LIN {X 0,Y 245.189,Z 1176.16,A -85,B 0,C 180,E1 20303.764,E2 20303.764} C_VEL
LIN {X 0,Y 259.827,Z 1145.905,A -85,B 0,C 180,E1 20307.743,E2 20307.743} C_VEL
LIN {X 0,Y 266.312,Z 1129.34,A -85,B 0,C 180,E1 20309.341,E2 20309.341} C_VEL
LIN {X 0,Y 263.727,Z 1110.426,A -85,B 0,C 180,E1 20314.736,E2 20314.736} C_VEL
LIN {X 0,Y 259.355,Z 1093.422,A -85,B 0,C 180,E1 20321.102,E2 20321.102} C_VEL
LIN {X 0,Y 255.054,Z 1081.089,A -85,B 0,C 180,E1 20327.942,E2 20327.942} C_VEL
LIN {X 0,Y 252.604,Z 1073.864,A -85,B 0,C 180,E1 20334.86,E2 20334.86} C_VEL
LIN {X 0,Y 252.397,Z 1073.391,A -85,B 0,C 180,E1 20342.571,E2 20342.571} C_VEL
LIN {X 0,Y 253.413,Z 1075.546,A -85,B 0,C 180,E1 20346.196,E2 20346.196} C_VEL
LIN {X 0,Y 256.742,Z 1083.33,A -85,B 0,C 180,E1 20352.41,E2 20352.41} C_VEL
LIN {X 0,Y 260.858,Z 1093.545,A -85,B 0,C 180,E1 20357.598,E2 20357.598} C_VEL
LIN {X 0,Y 262.032,Z 1131.057,A -85,B 0,C 180,E1 20365.325,E2 20365.325} C_VEL
LIN {X 0,Y 261.485,Z 1139.676,A -85,B 0,C 180,E1 20366.889,E2 20366.889} C_VEL
LIN {X 0,Y 247.883,Z 1174.599,A -85,B 0,C 180,E1 20370.279,E2 20370.279} C_VEL
LIN {X 0,Y 232.476,Z 1205.485,A -85,B 0,C 180,E1 20374.943,E2 20374.943} C_VEL
LIN {X 0,Y 216.883,Z 1231.951,A -85,B 0,C 180,E1 20380.998,E2 20380.998} C_VEL
LIN {X 0,Y 201.876,Z 1255.228,A -85,B 0,C 180,E1 20389.161,E2 20389.161} C_VEL
LIN {X 0,Y 190.362,Z 1273.058,A -85,B 0,C 180,E1 20398.994,E2 20398.994} C_VEL
LIN {X 0,Y 183.865,Z 1285.563,A -85,B 0,C 180,E1 20410.144,E2 20410.144} C_VEL
LIN {X 0,Y 182.005,Z 1292.009,A -85,B 0,C 180,E1 20420.464,E2 20420.464} C_VEL
LIN {X 0,Y 182.159,Z 1294.054,A -85,B 0,C 180,E1 20430.009,E2 20430.009} C_VEL
LIN {X 0,Y 182.027,Z 1292.019,A -85,B 0,C 180,E1 20439.553,E2 20439.553} C_VEL
LIN {X 0,Y 184.068,Z 1285.438,A -85,B 0,C 180,E1 20450.036,E2 20450.036} C_VEL
LIN {X 0,Y 190.629,Z 1273.108,A -85,B 0,C 180,E1 20460.978,E2 20460.978} C_VEL
LIN {X 0,Y 202.939,Z 1254.088,A -85,B 0,C 180,E1 20471.307,E2 20471.307} C_VEL
LIN {X 0,Y 218.493,Z 1230.096,A -85,B 0,C 180,E1 20479.452,E2 20479.452} C_VEL
LIN {X 0,Y 222.82,Z 1224.302,A -85,B 0,C 180,E1 20481.166,E2 20481.166} C_VEL
LIN {X 0,Y 227.633,Z 1220.781,A -85,B 0,C 180,E1 20482.716,E2 20482.716} C_VEL
LIN {X 0,Y 229.232,Z 1219.381,A -85,B 0,C 180,E1 20483.669,E2 20483.669} C_VEL
LIN {X 0,Y 212.52,Z 1224.351,A -85,B 0,C 180,E1 20490.196,E2 20490.196} C_VEL
LIN {X 0,Y 200.093,Z 1226.199,A -85,B 0,C 180,E1 20497.847,E2 20497.847} C_VEL
LIN {X 0,Y 190.04,Z 1223.798,A -85,B 0,C 180,E1 20508.55,E2 20508.55} C_VEL
LIN {X 0,Y 186.162,Z 1216.357,A -85,B 0,C 180,E1 20518.838,E2 20518.838} C_VEL
LIN {X 0,Y 186.218,Z 1204.944,A -85,B 0,C 180,E1 20528.151,E2 20528.151} C_VEL
LIN {X 0,Y 186.799,Z 1200.69,A -85,B 0,C 180,E1 20531.06,E2 20531.06} C_VEL
LIN {X 0,Y 208.406,Z 1192.088,A -85,B 0,C 180,E1 20545.748,E2 20545.748} C_VEL
LIN {X 0,Y 234.94,Z 1181.218,A -85,B 0,C 180,E1 20553.99,E2 20553.99} C_VEL
LIN {X 0,Y 244.119,Z 1176.975,A -85,B 0,C 180,E1 20555.967,E2 20555.967} C_VEL
LIN {X 0,Y 242.991,Z 1180.408,A -85,B 0,C 180,E1 20556.795,E2 20556.795} C_VEL
LIN {X 0,Y 235.158,Z 1193.598,A -85,B 0,C 180,E1 20559.308,E2 20559.308} C_VEL
LIN {X 0,Y 224.981,Z 1205.626,A -85,B 0,C 180,E1 20561.254,E2 20561.254} C_VEL
LIN {X 0,Y 214.6,Z 1216.631,A -85,B 0,C 180,E1 20563.537,E2 20563.537} C_VEL
LIN {X 0,Y 199.114,Z 1236.248,A -85,B 0,C 180,E1 20571.288,E2 20571.288} C_VEL
LIN {X 0,Y 186.349,Z 1251.331,A -85,B 0,C 180,E1 20580.92,E2 20580.92} C_VEL
LIN {X 0,Y 177.863,Z 1261.693,A -85,B 0,C 180,E1 20592.716,E2 20592.716} C_VEL
LIN {X 0,Y 175.408,Z 1265.154,A -85,B 0,C 180,E1 20600.083,E2 20600.083} C_VEL
LIN {X 0,Y 174.379,Z 1266.843,A -85,B 0,C 180,E1 20609.99,E2 20609.99} C_VEL
LIN {X 0,Y 175.404,Z 1265.113,A -85,B 0,C 180,E1 20619.898,E2 20619.898} C_VEL
LIN {X 0,Y 180.566,Z 1258.236,A -85,B 0,C 180,E1 20632.044,E2 20632.044} C_VEL
LIN {X 0,Y 191.47,Z 1245.156,A -85,B 0,C 180,E1 20643.473,E2 20643.473} C_VEL
LIN {X 0,Y 206.248,Z 1227.247,A -85,B 0,C 180,E1 20652.605,E2 20652.605} C_VEL
LIN {X 0,Y 223.911,Z 1203.483,A -85,B 0,C 180,E1 20660.002,E2 20660.002} C_VEL
LIN {X 0,Y 240.85,Z 1176.298,A -85,B 0,C 180,E1 20665.36,E2 20665.36} C_VEL
LIN {X 0,Y 255.839,Z 1146.194,A -85,B 0,C 180,E1 20669.271,E2 20669.271} C_VEL
LIN {X 0,Y 261.365,Z 1131.746,A -85,B 0,C 180,E1 20670.814,E2 20670.814} C_VEL
LIN {X 0,Y 259.219,Z 1113.75,A -85,B 0,C 180,E1 20676.341,E2 20676.341} C_VEL
LIN {X 0,Y 256.051,Z 1099.749,A -85,B 0,C 180,E1 20681.89,E2 20681.89} C_VEL
LIN {X 0,Y 252.505,Z 1087.186,A -85,B 0,C 180,E1 20689.138,E2 20689.138} C_VEL
LIN {X 0,Y 250.859,Z 1081.579,A -85,B 0,C 180,E1 20694.824,E2 20694.824} C_VEL
LIN {X 0,Y 250.784,Z 1081.139,A -85,B 0,C 180,E1 20702.587,E2 20702.587} C_VEL
LIN {X 0,Y 251.644,Z 1083.314,A -85,B 0,C 180,E1 20706.024,E2 20706.024} C_VEL
LIN {X 0,Y 254.452,Z 1090.646,A -85,B 0,C 180,E1 20711.98,E2 20711.98} C_VEL
LIN {X 0,Y 257.709,Z 1099.874,A -85,B 0,C 180,E1 20716.725,E2 20716.725} C_VEL
LIN {X 0,Y 257.468,Z 1137.249,A -85,B 0,C 180,E1 20724.682,E2 20724.682} C_VEL
LIN {X 0,Y 256.636,Z 1142.909,A -85,B 0,C 180,E1 20725.59,E2 20725.59} C_VEL
LIN {X 0,Y 242.493,Z 1176.928,A -85,B 0,C 180,E1 20728.999,E2 20728.999} C_VEL
LIN {X 0,Y 226.617,Z 1207.082,A -85,B 0,C 180,E1 20733.669,E2 20733.669} C_VEL
LIN {X 0,Y 209.266,Z 1234.843,A -85,B 0,C 180,E1 20740.333,E2 20740.333} C_VEL
LIN {X 0,Y 193.272,Z 1257.969,A -85,B 0,C 180,E1 20749.174,E2 20749.174} C_VEL
LIN {X 0,Y 181.334,Z 1275.631,A -85,B 0,C 180,E1 20760.056,E2 20760.056} C_VEL
LIN {X 0,Y 175.727,Z 1286.237,A -85,B 0,C 180,E1 20770.834,E2 20770.834} C_VEL
LIN {X 0,Y 174.128,Z 1291.399,A -85,B 0,C 180,E1 20780.028,E2 20780.028} C_VEL
LIN {X 0,Y 174.282,Z 1293.453,A -85,B 0,C 180,E1 20790.01,E2 20790.01} C_VEL
LIN {X 0,Y 174.15,Z 1291.41,A -85,B 0,C 180,E1 20799.99,E2 20799.99} C_VEL
LIN {X 0,Y 176.589,Z 1284.518,A -85,B 0,C 180,E1 20811.306,E2 20811.306} C_VEL
LIN {X 0,Y 184.769,Z 1270.858,A -85,B 0,C 180,E1 20823.466,E2 20823.466} C_VEL
LIN {X 0,Y 197.693,Z 1252.227,A -85,B 0,C 180,E1 20833.405,E2 20833.405} C_VEL
LIN {X 0,Y 215.557,Z 1227.057,A -85,B 0,C 180,E1 20841.973,E2 20841.973} C_VEL
LIN {X 0,Y 219.744,Z 1224.237,A -85,B 0,C 180,E1 20843.378,E2 20843.378} C_VEL
LIN {X 0,Y 218.871,Z 1224.206,A -85,B 0,C 180,E1 20844.125,E2 20844.125} C_VEL
LIN {X 0,Y 199.055,Z 1228.104,A -85,B 0,C 180,E1 20852.945,E2 20852.945} C_VEL
LIN {X 0,Y 188.026,Z 1227.701,A -85,B 0,C 180,E1 20861.275,E2 20861.275} C_VEL
LIN {X 0,Y 179.987,Z 1222.257,A -85,B 0,C 180,E1 20872.775,E2 20872.775} C_VEL
LIN {X 0,Y 178.093,Z 1211.877,A -85,B 0,C 180,E1 20883.642,E2 20883.642} C_VEL
LIN {X 0,Y 178.335,Z 1208.019,A -85,B 0,C 180,E1 20887.291,E2 20887.291} C_VEL
LIN {X 0,Y 198.763,Z 1199.468,A -85,B 0,C 180,E1 20904.327,E2 20904.327} C_VEL
LIN {X 0,Y 222.559,Z 1190.638,A -85,B 0,C 180,E1 20912.846,E2 20912.846} C_VEL
LIN {X 0,Y 234.82,Z 1185.521,A -85,B 0,C 180,E1 20915.778,E2 20915.778} C_VEL
LIN {X 0,Y 233.722,Z 1188.698,A -85,B 0,C 180,E1 20916.671,E2 20916.671} C_VEL
LIN {X 0,Y 216.238,Z 1214.459,A -85,B 0,C 180,E1 20922.87,E2 20922.87} C_VEL
LIN {X 0,Y 214.6,Z 1216.631,A -85,B 0,C 180,E1 20923.537,E2 20923.537} C_VEL
LIN {X 0,Y 204.086,Z 1226.81,A -85,B 0,C 180,E1 20926.208,E2 20926.208} C_VEL
LIN {X 0,Y 193.765,Z 1235.88,A -85,B 0,C 180,E1 20929.325,E2 20929.325} C_VEL
LIN {X 0,Y 179.406,Z 1251.939,A -85,B 0,C 180,E1 20939.679,E2 20939.679} C_VEL
LIN {X 0,Y 170.286,Z 1262.299,A -85,B 0,C 180,E1 20951.92,E2 20951.92} C_VEL
LIN {X 0,Y 166.738,Z 1266.954,A -85,B 0,C 180,E1 20964.534,E2 20964.534} C_VEL
LIN {X 0,Y 166.766,Z 1266.906,A -85,B 0,C 180,E1 20975.564,E2 20975.564} C_VEL
LIN {X 0,Y 170.295,Z 1262.227,A -85,B 0,C 180,E1 20988.058,E2 20988.058} C_VEL
LIN {X 0,Y 179.427,Z 1251.816,A -85,B 0,C 180,E1 21000.296,E2 21000.296} C_VEL
LIN {X 0,Y 193.837,Z 1235.62,A -85,B 0,C 180,E1 21010.682,E2 21010.682} C_VEL
LIN {X 0,Y 211.006,Z 1214.796,A -85,B 0,C 180,E1 21018.659,E2 21018.659} C_VEL
LIN {X 0,Y 229.31,Z 1188.648,A -85,B 0,C 180,E1 21024.922,E2 21024.922} C_VEL
LIN {X 0,Y 245.601,Z 1159.936,A -85,B 0,C 180,E1 21029.327,E2 21029.327} C_VEL
LIN {X 0,Y 256.523,Z 1135.753,A -85,B 0,C 180,E1 21031.929,E2 21031.929} C_VEL
LIN {X 0,Y 255.032,Z 1118.805,A -85,B 0,C 180,E1 21037.383,E2 21037.383} C_VEL
LIN {X 0,Y 252.373,Z 1104.64,A -85,B 0,C 180,E1 21043.411,E2 21043.411} C_VEL
LIN {X 0,Y 249.75,Z 1093.879,A -85,B 0,C 180,E1 21050.217,E2 21050.217} C_VEL
LIN {X 0,Y 248.747,Z 1089.066,A -85,B 0,C 180,E1 21055.652,E2 21055.652} C_VEL
LIN {X 0,Y 249.002,Z 1088.918,A -85,B 0,C 180,E1 21063.04,E2 21063.04} C_VEL
LIN {X 0,Y 249.794,Z 1091.622,A -85,B 0,C 180,E1 21066.395,E2 21066.395} C_VEL
LIN {X 0,Y 252.674,Z 1099.304,A -85,B 0,C 180,E1 21072.613,E2 21072.613} C_VEL
LIN {X 0,Y 254.53,Z 1105.732,A -85,B 0,C 180,E1 21075.743,E2 21075.743} C_VEL
LIN {X 0,Y 252.921,Z 1141.925,A -85,B 0,C 180,E1 21083.688,E2 21083.688} C_VEL
LIN {X 0,Y 251.045,Z 1148.161,A -85,B 0,C 180,E1 21084.433,E2 21084.433} C_VEL
LIN {X 0,Y 235.684,Z 1182.305,A -85,B 0,C 180,E1 21088.041,E2 21088.041} C_VEL
LIN {X 0,Y 218.408,Z 1212.526,A -85,B 0,C 180,E1 21093.11,E2 21093.11} C_VEL
LIN {X 0,Y 200.991,Z 1238.491,A -85,B 0,C 180,E1 21099.929,E2 21099.929} C_VEL
LIN {X 0,Y 184.644,Z 1260.616,A -85,B 0,C 180,E1 21109.182,E2 21109.182} C_VEL
LIN {X 0,Y 173.275,Z 1276.452,A -85,B 0,C 180,E1 21119.989,E2 21119.989} C_VEL
LIN {X 0,Y 167.402,Z 1287.158,A -85,B 0,C 180,E1 21132.304,E2 21132.304} C_VEL
LIN {X 0,Y 166.257,Z 1290.788,A -85,B 0,C 180,E1 21139.551,E2 21139.551} C_VEL
LIN {X 0,Y 166.389,Z 1292.85,A -85,B 0,C 180,E1 21150.01,E2 21150.01} C_VEL
LIN {X 0,Y 166.279,Z 1290.8,A -85,B 0,C 180,E1 21160.468,E2 21160.468} C_VEL
LIN {X 0,Y 169.039,Z 1283.899,A -85,B 0,C 180,E1 21172.308,E2 21172.308} C_VEL
LIN {X 0,Y 176.763,Z 1271.861,A -85,B 0,C 180,E1 21183.716,E2 21183.716} C_VEL
LIN {X 0,Y 190.692,Z 1253.112,A -85,B 0,C 180,E1 21194.454,E2 21194.454} C_VEL
LIN {X 0,Y 208.282,Z 1229.52,A -85,B 0,C 180,E1 21202.856,E2 21202.856} C_VEL
LIN {X 0,Y 209.933,Z 1228.085,A -85,B 0,C 180,E1 21204.052,E2 21204.052} C_VEL
LIN {X 0,Y 192.381,Z 1230.422,A -85,B 0,C 180,E1 21211.925,E2 21211.925} C_VEL
LIN {X 0,Y 180.743,Z 1229.449,A -85,B 0,C 180,E1 21220.491,E2 21220.491} C_VEL
LIN {X 0,Y 172.225,Z 1223.336,A -85,B 0,C 180,E1 21232.447,E2 21232.447} C_VEL
LIN {X 0,Y 170.257,Z 1215.578,A -85,B 0,C 180,E1 21241.269,E2 21241.269} C_VEL
LIN {X 0,Y 186.699,Z 1207.359,A -85,B 0,C 180,E1 21261.327,E2 21261.327} C_VEL
LIN {X 0,Y 212.387,Z 1198.52,A -85,B 0,C 180,E1 21272.197,E2 21272.197} C_VEL
LIN {X 0,Y 225.811,Z 1193.374,A -85,B 0,C 180,E1 21275.661,E2 21275.661} C_VEL
LIN {X 0,Y 223.008,Z 1198.447,A -85,B 0,C 180,E1 21276.956,E2 21276.956} C_VEL
LIN {X 0,Y 205.444,Z 1221.95,A -85,B 0,C 180,E1 21283.522,E2 21283.522} C_VEL
LIN {X 0,Y 193.765,Z 1235.88,A -85,B 0,C 180,E1 21289.325,E2 21289.325} C_VEL
LIN {X 0,Y 183.692,Z 1243.998,A -85,B 0,C 180,E1 21292.93,E2 21292.93} C_VEL
LIN {X 0,Y 174.018,Z 1250.991,A -85,B 0,C 180,E1 21297.05,E2 21297.05} C_VEL
LIN {X 0,Y 164.217,Z 1261.318,A -85,B 0,C 180,E1 21308.423,E2 21308.423} C_VEL
LIN {X 0,Y 159.862,Z 1266.359,A -85,B 0,C 180,E1 21319.107,E2 21319.107} C_VEL
LIN {X 0,Y 158.63,Z 1268.045,A -85,B 0,C 180,E1 21329.989,E2 21329.989} C_VEL
LIN {X 0,Y 159.855,Z 1266.319,A -85,B 0,C 180,E1 21340.872,E2 21340.872} C_VEL
LIN {X 0,Y 165.373,Z 1259.988,A -85,B 0,C 180,E1 21353.343,E2 21353.343} C_VEL
LIN {X 0,Y 176.842,Z 1248.03,A -85,B 0,C 180,E1 21365.158,E2 21365.158} C_VEL
LIN {X 0,Y 192.75,Z 1230.808,A -85,B 0,C 180,E1 21374.787,E2 21374.787} C_VEL
LIN {X 0,Y 210.471,Z 1209.398,A -85,B 0,C 180,E1 21382.05,E2 21382.05} C_VEL
LIN {X 0,Y 229.446,Z 1182.101,A -85,B 0,C 180,E1 21387.85,E2 21387.85} C_VEL
LIN {X 0,Y 246.322,Z 1151.212,A -85,B 0,C 180,E1 21392.003,E2 21392.003} C_VEL
LIN {X 0,Y 251.68,Z 1138.595,A -85,B 0,C 180,E1 21393.424,E2 21393.424} C_VEL
LIN {X 0,Y 250.651,Z 1121.653,A -85,B 0,C 180,E1 21399.288,E2 21399.288} C_VEL
LIN {X 0,Y 248.464,Z 1107.88,A -85,B 0,C 180,E1 21405.942,E2 21405.942} C_VEL
LIN {X 0,Y 246.888,Z 1100.12,A -85,B 0,C 180,E1 21411.765,E2 21411.765} C_VEL
LIN {X 0,Y 246.49,Z 1096.612,A -85,B 0,C 180,E1 21415.798,E2 21415.798} C_VEL
LIN {X 0,Y 246.762,Z 1096.421,A -85,B 0,C 180,E1 21422.629,E2 21422.629} C_VEL
LIN {X 0,Y 247.472,Z 1099.22,A -85,B 0,C 180,E1 21426.236,E2 21426.236} C_VEL
LIN {X 0,Y 249.649,Z 1105.719,A -85,B 0,C 180,E1 21431.605,E2 21431.605} C_VEL
LIN {X 0,Y 251.154,Z 1111.895,A -85,B 0,C 180,E1 21434.84,E2 21434.84} C_VEL
LIN {X 0,Y 248.303,Z 1146.097,A -85,B 0,C 180,E1 21442.572,E2 21442.572} C_VEL
LIN {X 0,Y 232.505,Z 1180.722,A -85,B 0,C 180,E1 21446.145,E2 21446.145} C_VEL
LIN {X 0,Y 215.352,Z 1209.958,A -85,B 0,C 180,E1 21450.877,E2 21450.877} C_VEL
LIN {X 0,Y 197.136,Z 1236.072,A -85,B 0,C 180,E1 21457.503,E2 21457.503} C_VEL
LIN {X 0,Y 179.845,Z 1258.353,A -85,B 0,C 180,E1 21466.587,E2 21466.587} C_VEL
LIN {X 0,Y 166.334,Z 1275.657,A -85,B 0,C 180,E1 21478.418,E2 21478.418} C_VEL
LIN {X 0,Y 159.887,Z 1286.096,A -85,B 0,C 180,E1 21490.695,E2 21490.695} C_VEL
LIN {X 0,Y 158.393,Z 1290.177,A -85,B 0,C 180,E1 21499.026,E2 21499.026} C_VEL
LIN {X 0,Y 158.511,Z 1292.249,A -85,B 0,C 180,E1 21510.011,E2 21510.011} C_VEL
LIN {X 0,Y 158.417,Z 1290.189,A -85,B 0,C 180,E1 21520.994,E2 21520.994} C_VEL
LIN {X 0,Y 161.528,Z 1283.279,A -85,B 0,C 180,E1 21533.405,E2 21533.405} C_VEL
LIN {X 0,Y 169.964,Z 1271.234,A -85,B 0,C 180,E1 21545.26,E2 21545.26} C_VEL
LIN {X 0,Y 184.925,Z 1252.491,A -85,B 0,C 180,E1 21556.234,E2 21556.234} C_VEL
LIN {X 0,Y 200.873,Z 1231.575,A -85,B 0,C 180,E1 21563.994,E2 21563.994} C_VEL
LIN {X 0,Y 179.115,Z 1232.266,A -85,B 0,C 180,E1 21575.087,E2 21575.087} C_VEL
LIN {X 0,Y 167.187,Z 1227.702,A -85,B 0,C 180,E1 21586.959,E2 21586.959} C_VEL
LIN {X 0,Y 163.61,Z 1223.156,A -85,B 0,C 180,E1 21594.707,E2 21594.707} C_VEL
LIN {X 0,Y 184.744,Z 1211.533,A -85,B 0,C 180,E1 21624.103,E2 21624.103} C_VEL
LIN {X 0,Y 212.713,Z 1202.262,A -85,B 0,C 180,E1 21634.575,E2 21634.575} C_VEL
LIN {X 0,Y 216.482,Z 1200.929,A -85,B 0,C 180,E1 21635.529,E2 21635.529} C_VEL
LIN {X 0,Y 199.29,Z 1223.447,A -85,B 0,C 180,E1 21642.195,E2 21642.195} C_VEL
LIN {X 0,Y 183.326,Z 1241.297,A -85,B 0,C 180,E1 21650.349,E2 21650.349} C_VEL
LIN {X 0,Y 174.018,Z 1250.991,A -85,B 0,C 180,E1 21657.05,E2 21657.05} C_VEL
LIN {X 0,Y 165.048,Z 1256.934,A -85,B 0,C 180,E1 21661.74,E2 21661.74} C_VEL
LIN {X 0,Y 157.034,Z 1261.713,A -85,B 0,C 180,E1 21667.034,E2 21667.034} C_VEL
LIN {X 0,Y 152.089,Z 1266.964,A -85,B 0,C 180,E1 21678.543,E2 21678.543} C_VEL
LIN {X 0,Y 150.759,Z 1268.646,A -85,B 0,C 180,E1 21689.989,E2 21689.989} C_VEL
LIN {X 0,Y 152.081,Z 1266.924,A -85,B 0,C 180,E1 21701.435,E2 21701.435} C_VEL
LIN {X 0,Y 157.886,Z 1260.8,A -85,B 0,C 180,E1 21714.181,E2 21714.181} C_VEL
LIN {X 0,Y 170.386,Z 1248.638,A -85,B 0,C 180,E1 21726.702,E2 21726.702} C_VEL
LIN {X 0,Y 187.178,Z 1231.415,A -85,B 0,C 180,E1 21736.505,E2 21736.505} C_VEL
LIN {X 0,Y 206.521,Z 1208.947,A -85,B 0,C 180,E1 21744.083,E2 21744.083} C_VEL
LIN {X 0,Y 226.033,Z 1181.588,A -85,B 0,C 180,E1 21749.725,E2 21749.725} C_VEL
LIN {X 0,Y 242.637,Z 1151.967,A -85,B 0,C 180,E1 21753.632,E2 21753.632} C_VEL
LIN {X 0,Y 246.974,Z 1142.389,A -85,B 0,C 180,E1 21754.68,E2 21754.68} C_VEL
LIN {X 0,Y 246.55,Z 1125.822,A -85,B 0,C 180,E1 21760.795,E2 21760.795} C_VEL
LIN {X 0,Y 244.976,Z 1112.678,A -85,B 0,C 180,E1 21767.709,E2 21767.709} C_VEL
LIN {X 0,Y 244.18,Z 1104.268,A -85,B 0,C 180,E1 21775.058,E2 21775.058} C_VEL
LIN {X 0,Y 244.112,Z 1103.348,A -85,B 0,C 180,E1 21780.001,E2 21780.001} C_VEL
LIN {X 0,Y 244.781,Z 1105.243,A -85,B 0,C 180,E1 21784.697,E2 21784.697} C_VEL
LIN {X 0,Y 246.87,Z 1113.425,A -85,B 0,C 180,E1 21791.54,E2 21791.54} C_VEL
LIN {X 0,Y 247.813,Z 1116.958,A -85,B 0,C 180,E1 21793.604,E2 21793.604} C_VEL
LIN {X 0,Y 243.764,Z 1149.572,A -85,B 0,C 180,E1 21801.198,E2 21801.198} C_VEL
LIN {X 0,Y 227.344,Z 1183.103,A -85,B 0,C 180,E1 21804.713,E2 21804.713} C_VEL
LIN {X 0,Y 209.921,Z 1211.287,A -85,B 0,C 180,E1 21809.368,E2 21809.368} C_VEL
LIN {X 0,Y 190.906,Z 1237.147,A -85,B 0,C 180,E1 21816.103,E2 21816.103} C_VEL
LIN {X 0,Y 172.532,Z 1259.362,A -85,B 0,C 180,E1 21825.609,E2 21825.609} C_VEL
LIN {X 0,Y 159.501,Z 1274.907,A -85,B 0,C 180,E1 21836.755,E2 21836.755} C_VEL
LIN {X 0,Y 152.238,Z 1285.475,A -85,B 0,C 180,E1 21849.683,E2 21849.683} C_VEL
LIN {X 0,Y 150.544,Z 1289.566,A -85,B 0,C 180,E1 21858.446,E2 21858.446} C_VEL
LIN {X 0,Y 150.618,Z 1291.647,A -85,B 0,C 180,E1 21870.011,E2 21870.011} C_VEL
LIN {X 0,Y 150.595,Z 1289.581,A -85,B 0,C 180,E1 21881.572,E2 21881.572} C_VEL
LIN {X 0,Y 154.087,Z 1282.658,A -85,B 0,C 180,E1 21894.608,E2 21894.608} C_VEL
LIN {X 0,Y 163.325,Z 1270.61,A -85,B 0,C 180,E1 21906.924,E2 21906.924} C_VEL
LIN {X 0,Y 179.675,Z 1251.451,A -85,B 0,C 180,E1 21918.315,E2 21918.315} C_VEL
LIN {X 0,Y 191.17,Z 1237.393,A -85,B 0,C 180,E1 21923.743,E2 21923.743} C_VEL
LIN {X 0,Y 191.403,Z 1236.168,A -85,B 0,C 180,E1 21924.383,E2 21924.383} C_VEL
LIN {X 0,Y 166.271,Z 1232.825,A -85,B 0,C 180,E1 21938.714,E2 21938.714} C_VEL
LIN {X 0,Y 172.135,Z 1218.899,A -85,B 0,C 180,E1 21980.525,E2 21980.525} C_VEL
LIN {X 0,Y 206.98,Z 1208.549,A -85,B 0,C 180,E1 21995.676,E2 21995.676} C_VEL
LIN {X 0,Y 188.21,Z 1230.468,A -85,B 0,C 180,E1 22002.967,E2 22002.967} C_VEL
LIN {X 0,Y 171.707,Z 1247.39,A -85,B 0,C 180,E1 22012.269,E2 22012.269} C_VEL
LIN {X 0,Y 159.314,Z 1259.468,A -85,B 0,C 180,E1 22023.79,E2 22023.79} C_VEL
LIN {X 0,Y 157.034,Z 1261.713,A -85,B 0,C 180,E1 22027.034,E2 22027.034} C_VEL
LIN {X 0,Y 152.147,Z 1264.589,A -85,B 0,C 180,E1 22031.423,E2 22031.423} C_VEL
LIN {X 0,Y 144.275,Z 1267.687,A -85,B 0,C 180,E1 22038.394,E2 22038.394} C_VEL
LIN {X 0,Y 143.942,Z 1267.845,A -85,B 0,C 180,E1 22039.258,E2 22039.258} C_VEL
LIN {X 0,Y 142.879,Z 1269.247,A -85,B 0,C 180,E1 22049.988,E2 22049.988} C_VEL
LIN {X 0,Y 144.338,Z 1267.528,A -85,B 0,C 180,E1 22062.058,E2 22062.058} C_VEL
LIN {X 0,Y 151.066,Z 1261.049,A -85,B 0,C 180,E1 22075.979,E2 22075.979} C_VEL
LIN {X 0,Y 163.868,Z 1249.429,A -85,B 0,C 180,E1 22088.23,E2 22088.23} C_VEL
LIN {X 0,Y 182.191,Z 1231.606,A -85,B 0,C 180,E1 22098.505,E2 22098.505} C_VEL
LIN {X 0,Y 202.17,Z 1209.308,A -85,B 0,C 180,E1 22105.971,E2 22105.971} C_VEL
LIN {X 0,Y 222.848,Z 1181.069,A -85,B 0,C 180,E1 22111.665,E2 22111.665} C_VEL
LIN {X 0,Y 239.933,Z 1151.141,A -85,B 0,C 180,E1 22115.476,E2 22115.476} C_VEL
LIN {X 0,Y 242.38,Z 1145.603,A -85,B 0,C 180,E1 22116.201,E2 22116.201} C_VEL
LIN {X 0,Y 242.5,Z 1131.082,A -85,B 0,C 180,E1 22121.874,E2 22121.874} C_VEL
LIN {X 0,Y 241.778,Z 1119.443,A -85,B 0,C 180,E1 22128.298,E2 22128.298} C_VEL
LIN {X 0,Y 241.447,Z 1112.003,A -85,B 0,C 180,E1 22135.002,E2 22135.002} C_VEL
LIN {X 0,Y 241.542,Z 1110.826,A -85,B 0,C 180,E1 22140.001,E2 22140.001} C_VEL
LIN {X 0,Y 242.11,Z 1112.508,A -85,B 0,C 180,E1 22144.329,E2 22144.329} C_VEL
LIN {X 0,Y 243.898,Z 1121.412,A -85,B 0,C 180,E1 22151.682,E2 22151.682} C_VEL
LIN {X 0,Y 244.152,Z 1124.422,A -85,B 0,C 180,E1 22153.071,E2 22153.071} C_VEL
LIN {X 0,Y 239.703,Z 1151.507,A -85,B 0,C 180,E1 22159.538,E2 22159.538} C_VEL
LIN {X 0,Y 222.574,Z 1185.04,A -85,B 0,C 180,E1 22163.16,E2 22163.16} C_VEL
LIN {X 0,Y 203.297,Z 1214.544,A -85,B 0,C 180,E1 22168.183,E2 22168.183} C_VEL
LIN {X 0,Y 182.848,Z 1240.489,A -85,B 0,C 180,E1 22175.422,E2 22175.422} C_VEL
LIN {X 0,Y 164.862,Z 1260.757,A -85,B 0,C 180,E1 22184.829,E2 22184.829} C_VEL
LIN {X 0,Y 151.259,Z 1275.954,A -85,B 0,C 180,E1 22196.734,E2 22196.734} C_VEL
LIN {X 0,Y 144.011,Z 1285.962,A -85,B 0,C 180,E1 22210.568,E2 22210.568} C_VEL
LIN {X 0,Y 142.346,Z 1290.459,A -85,B 0,C 180,E1 22223.926,E2 22223.926} C_VEL
LIN {X 0,Y 142.719,Z 1291.044,A -85,B 0,C 180,E1 22230.012,E2 22230.012} C_VEL
LIN {X 0,Y 142.748,Z 1288.97,A -85,B 0,C 180,E1 22242.218,E2 22242.218} C_VEL
LIN {X 0,Y 146.687,Z 1282.035,A -85,B 0,C 180,E1 22255.939,E2 22255.939} C_VEL
LIN {X 0,Y 157.741,Z 1269.013,A -85,B 0,C 180,E1 22269.53,E2 22269.53} C_VEL
LIN {X 0,Y 175.278,Z 1249.74,A -85,B 0,C 180,E1 22280.807,E2 22280.807} C_VEL
LIN {X 0,Y 182.492,Z 1240.72,A -85,B 0,C 180,E1 22284.633,E2 22284.633} C_VEL
LIN {X 0,Y 155.611,Z 1236.116,A -85,B 0,C 180,E1 22303.087,E2 22303.087} C_VEL
LIN {X 0,Y 169.698,Z 1222.695,A -85,B 0,C 180,E1 22343.586,E2 22343.586} C_VEL
LIN {X 0,Y 196.981,Z 1214.875,A -85,B 0,C 180,E1 22355.045,E2 22355.045} C_VEL
LIN {X 0,Y 193.49,Z 1219.675,A -85,B 0,C 180,E1 22356.912,E2 22356.912} C_VEL
LIN {X 0,Y 173.323,Z 1240.642,A -85,B 0,C 180,E1 22365.837,E2 22365.837} C_VEL
LIN {X 0,Y 157.722,Z 1255.028,A -85,B 0,C 180,E1 22376.61,E2 22376.61} C_VEL
LIN {X 0,Y 147.832,Z 1264.113,A -85,B 0,C 180,E1 22389.055,E2 22389.055} C_VEL
LIN {X 0,Y 143.942,Z 1267.845,A -85,B 0,C 180,E1 22399.258,E2 22399.258} C_VEL
LIN {X 0,Y 140.501,Z 1269.085,A -85,B 0,C 180,E1 22404.328,E2 22404.328} C_VEL
LIN {X 0,Y 134.969,Z 1269.615,A -85,B 0,C 180,E1 22413.208,E2 22413.208} C_VEL
LIN {X 0,Y 137.544,Z 1267.205,A -85,B 0,C 180,E1 22425.907,E2 22425.907} C_VEL
LIN {X 0,Y 146.933,Z 1259.116,A -85,B 0,C 180,E1 22440.885,E2 22440.885} C_VEL
LIN {X 0,Y 161.652,Z 1246.54,A -85,B 0,C 180,E1 22452.58,E2 22452.58} C_VEL
LIN {X 0,Y 181.356,Z 1227.92,A -85,B 0,C 180,E1 22462.216,E2 22462.216} C_VEL
LIN {X 0,Y 202.141,Z 1204.714,A -85,B 0,C 180,E1 22469.134,E2 22469.134} C_VEL
LIN {X 0,Y 222.14,Z 1177.196,A -85,B 0,C 180,E1 22474.155,E2 22474.155} C_VEL
LIN {X 0,Y 237.837,Z 1149.178,A -85,B 0,C 180,E1 22477.626,E2 22477.626} C_VEL
LIN {X 0,Y 238.482,Z 1135.322,A -85,B 0,C 180,E1 22483.456,E2 22483.456} C_VEL
LIN {X 0,Y 238.316,Z 1124.631,A -85,B 0,C 180,E1 22489.973,E2 22489.973} C_VEL
LIN {X 0,Y 238.487,Z 1118.808,A -85,B 0,C 180,E1 22496.373,E2 22496.373} C_VEL
LIN {X 0,Y 238.695,Z 1118.181,A -85,B 0,C 180,E1 22500.001,E2 22500.001} C_VEL
LIN {X 0,Y 239.151,Z 1119.336,A -85,B 0,C 180,E1 22503.618,E2 22503.618} C_VEL
LIN {X 0,Y 240.466,Z 1127.7,A -85,B 0,C 180,E1 22510.851,E2 22510.851} C_VEL
LIN {X 0,Y 240.406,Z 1130.835,A -85,B 0,C 180,E1 22512.231,E2 22512.231} C_VEL
LIN {X 0,Y 235.396,Z 1154.888,A -85,B 0,C 180,E1 22518.123,E2 22518.123} C_VEL
LIN {X 0,Y 217.201,Z 1188.248,A -85,B 0,C 180,E1 22521.701,E2 22521.701} C_VEL
LIN {X 0,Y 196.658,Z 1217.658,A -85,B 0,C 180,E1 22526.928,E2 22526.928} C_VEL
LIN {X 0,Y 176.654,Z 1241.573,A -85,B 0,C 180,E1 22533.894,E2 22533.894} C_VEL
LIN {X 0,Y 157.206,Z 1262.15,A -85,B 0,C 180,E1 22543.966,E2 22543.966} C_VEL
LIN {X 0,Y 143.248,Z 1276.714,A -85,B 0,C 180,E1 22556.436,E2 22556.436} C_VEL
LIN {X 0,Y 136.068,Z 1285.904,A -85,B 0,C 180,E1 22570.579,E2 22570.579} C_VEL
LIN {X 0,Y 134.439,Z 1289.851,A -85,B 0,C 180,E1 22583.568,E2 22583.568} C_VEL
LIN {X 0,Y 134.824,Z 1290.441,A -85,B 0,C 180,E1 22590.012,E2 22590.012} C_VEL
LIN {X 0,Y 134.914,Z 1288.358,A -85,B 0,C 180,E1 22602.94,E2 22602.94} C_VEL
LIN {X 0,Y 139.379,Z 1281.422,A -85,B 0,C 180,E1 22617.395,E2 22617.395} C_VEL
LIN {X 0,Y 151.197,Z 1268.698,A -85,B 0,C 180,E1 22631.244,E2 22631.244} C_VEL
LIN {X 0,Y 168.526,Z 1250.931,A -85,B 0,C 180,E1 22642.155,E2 22642.155} C_VEL
LIN {X 0,Y 172.973,Z 1246.131,A -85,B 0,C 180,E1 22644.254,E2 22644.254} C_VEL
LIN {X 0,Y 173.089,Z 1244.848,A -85,B 0,C 180,E1 22645.202,E2 22645.202} C_VEL
LIN {X 0,Y 146.179,Z 1239.056,A -85,B 0,C 180,E1 22668.084,E2 22668.084} C_VEL
LIN {X 0,Y 167.723,Z 1226.36,A -85,B 0,C 180,E1 22706.732,E2 22706.732} C_VEL
LIN {X 0,Y 187.644,Z 1220.987,A -85,B 0,C 180,E1 22714.92,E2 22714.92} C_VEL
LIN {X 0,Y 183.788,Z 1225.578,A -85,B 0,C 180,E1 22716.802,E2 22716.802} C_VEL
LIN {X 0,Y 163.569,Z 1244.977,A -85,B 0,C 180,E1 22726.202,E2 22726.202} C_VEL
LIN {X 0,Y 146.909,Z 1259.209,A -85,B 0,C 180,E1 22739.083,E2 22739.083} C_VEL
LIN {X 0,Y 137.547,Z 1267.258,A -85,B 0,C 180,E1 22754.068,E2 22754.068} C_VEL
LIN {X 0,Y 135.319,Z 1269.409,A -85,B 0,C 180,E1 22763.585,E2 22763.585} C_VEL
LIN {X 0,Y 134.969,Z 1269.615,A -85,B 0,C 180,E1 22773.208,E2 22773.208} C_VEL
LIN {X 0,Y 133.078,Z 1269.268,A -85,B 0,C 180,E1 22778.759,E2 22778.759} C_VEL
LIN {X 0,Y 130.202,Z 1267.651,A -85,B 0,C 180,E1 22787.318,E2 22787.318} C_VEL
LIN {X 0,Y 130.51,Z 1267.332,A -85,B 0,C 180,E1 22788.27,E2 22788.27} C_VEL
LIN {X 0,Y 141.555,Z 1258.646,A -85,B 0,C 180,E1 22804.019,E2 22804.019} C_VEL
LIN {X 0,Y 157.94,Z 1245.422,A -85,B 0,C 180,E1 22815.759,E2 22815.759} C_VEL
LIN {X 0,Y 179.175,Z 1225.966,A -85,B 0,C 180,E1 22825.186,E2 22825.186} C_VEL
LIN {X 0,Y 201.042,Z 1201.921,A -85,B 0,C 180,E1 22831.864,E2 22831.864} C_VEL
LIN {X 0,Y 221.821,Z 1173.081,A -85,B 0,C 180,E1 22836.676,E2 22836.676} C_VEL
LIN {X 0,Y 233.366,Z 1152.726,A -85,B 0,C 180,E1 22839.139,E2 22839.139} C_VEL
LIN {X 0,Y 234.571,Z 1139.666,A -85,B 0,C 180,E1 22845.09,E2 22845.09} C_VEL
LIN {X 0,Y 234.91,Z 1131.109,A -85,B 0,C 180,E1 22850.76,E2 22850.76} C_VEL
LIN {X 0,Y 235.34,Z 1126.177,A -85,B 0,C 180,E1 22856.325,E2 22856.325} C_VEL
LIN {X 0,Y 235.667,Z 1125.48,A -85,B 0,C 180,E1 22860.001,E2 22860.001} C_VEL
LIN {X 0,Y 236.045,Z 1126.826,A -85,B 0,C 180,E1 22863.666,E2 22863.666} C_VEL
LIN {X 0,Y 236.863,Z 1134.048,A -85,B 0,C 180,E1 22870.09,E2 22870.09} C_VEL
LIN {X 0,Y 236.607,Z 1137.089,A -85,B 0,C 180,E1 22871.339,E2 22871.339} C_VEL
LIN {X 0,Y 231.052,Z 1158.387,A -85,B 0,C 180,E1 22876.574,E2 22876.574} C_VEL
LIN {X 0,Y 211.967,Z 1191.153,A -85,B 0,C 180,E1 22880.162,E2 22880.162} C_VEL
LIN {X 0,Y 190.578,Z 1220.111,A -85,B 0,C 180,E1 22885.451,E2 22885.451} C_VEL
LIN {X 0,Y 168.28,Z 1245.091,A -85,B 0,C 180,E1 22893.219,E2 22893.219} C_VEL
LIN {X 0,Y 149.602,Z 1263.403,A -85,B 0,C 180,E1 22903.019,E2 22903.019} C_VEL
LIN {X 0,Y 135.22,Z 1277.31,A -85,B 0,C 180,E1 22916.097,E2 22916.097} C_VEL
LIN {X 0,Y 128.189,Z 1285.661,A -85,B 0,C 180,E1 22930.343,E2 22930.343} C_VEL
LIN {X 0,Y 126.529,Z 1289.243,A -85,B 0,C 180,E1 22943.164,E2 22943.164} C_VEL
LIN {X 0,Y 126.92,Z 1289.838,A -85,B 0,C 180,E1 22950.013,E2 22950.013} C_VEL
LIN {X 0,Y 127.101,Z 1287.745,A -85,B 0,C 180,E1 22963.75,E2 22963.75} C_VEL
LIN {X 0,Y 131.28,Z 1281.824,A -85,B 0,C 180,E1 22977.388,E2 22977.388} C_VEL
LIN {X 0,Y 142.876,Z 1270.137,A -85,B 0,C 180,E1 22991.582,E2 22991.582} C_VEL
LIN {X 0,Y 161.975,Z 1251.881,A -85,B 0,C 180,E1 23003.672,E2 23003.672} C_VEL
LIN {X 0,Y 164.326,Z 1248.754,A -85,B 0,C 180,E1 23005.427,E2 23005.427} C_VEL
LIN {X 0,Y 139.657,Z 1243.319,A -85,B 0,C 180,E1 23027.519,E2 23027.519} C_VEL
LIN {X 0,Y 161.906,Z 1230.917,A -85,B 0,C 180,E1 23067.773,E2 23067.773} C_VEL
LIN {X 0,Y 178.054,Z 1226.781,A -85,B 0,C 180,E1 23074.702,E2 23074.702} C_VEL
LIN {X 0,Y 165.778,Z 1238.716,A -85,B 0,C 180,E1 23080.197,E2 23080.197} C_VEL
LIN {X 0,Y 146.375,Z 1254.97,A -85,B 0,C 180,E1 23091.774,E2 23091.774} C_VEL
LIN {X 0,Y 133.101,Z 1265.325,A -85,B 0,C 180,E1 23106.607,E2 23106.607} C_VEL
LIN {X 0,Y 128.925,Z 1268.772,A -85,B 0,C 180,E1 23116.448,E2 23116.448} C_VEL
LIN {X 0,Y 127.143,Z 1270.448,A -85,B 0,C 180,E1 23129.987,E2 23129.987} C_VEL
LIN {X 0,Y 128.917,Z 1268.735,A -85,B 0,C 180,E1 23143.526,E2 23143.526} C_VEL
LIN {X 0,Y 130.51,Z 1267.332,A -85,B 0,C 180,E1 23148.27,E2 23148.27} C_VEL
LIN {X 0,Y 130.911,Z 1265.43,A -85,B 0,C 180,E1 23153.968,E2 23153.968} C_VEL
LIN {X 0,Y 131.747,Z 1261.672,A -85,B 0,C 180,E1 23162.483,E2 23162.483} C_VEL
LIN {X 0,Y 132.451,Z 1261.081,A -85,B 0,C 180,E1 23163.354,E2 23163.354} C_VEL
LIN {X 0,Y 150.279,Z 1247.758,A -85,B 0,C 180,E1 23176.704,E2 23176.704} C_VEL
LIN {X 0,Y 172.078,Z 1229.13,A -85,B 0,C 180,E1 23186.402,E2 23186.402} C_VEL
LIN {X 0,Y 194.472,Z 1205.919,A -85,B 0,C 180,E1 23193.154,E2 23193.154} C_VEL
LIN {X 0,Y 215.7,Z 1178.392,A -85,B 0,C 180,E1 23197.948,E2 23197.948} C_VEL
LIN {X 0,Y 228.316,Z 1158.098,A -85,B 0,C 180,E1 23200.334,E2 23200.334} C_VEL
LIN {X 0,Y 230.033,Z 1149.576,A -85,B 0,C 180,E1 23203.813,E2 23203.813} C_VEL
LIN {X 0,Y 231.245,Z 1138.058,A -85,B 0,C 180,E1 23211.042,E2 23211.042} C_VEL
LIN {X 0,Y 231.998,Z 1133.489,A -85,B 0,C 180,E1 23216.272,E2 23216.272} C_VEL
LIN {X 0,Y 232.426,Z 1132.71,A -85,B 0,C 180,E1 23220.001,E2 23220.001} C_VEL
LIN {X 0,Y 232.747,Z 1136.013,A -85,B 0,C 180,E1 23225.581,E2 23225.581} C_VEL
LIN {X 0,Y 233.109,Z 1141.098,A -85,B 0,C 180,E1 23229.784,E2 23229.784} C_VEL
LIN {X 0,Y 227.125,Z 1161.072,A -85,B 0,C 180,E1 23234.921,E2 23234.921} C_VEL
LIN {X 0,Y 207.694,Z 1192.862,A -85,B 0,C 180,E1 23238.386,E2 23238.386} C_VEL
LIN {X 0,Y 185.351,Z 1221.706,A -85,B 0,C 180,E1 23243.69,E2 23243.69} C_VEL
LIN {X 0,Y 161.998,Z 1246.264,A -85,B 0,C 180,E1 23251.561,E2 23251.561} C_VEL
LIN {X 0,Y 142.027,Z 1264.585,A -85,B 0,C 180,E1 23261.965,E2 23261.965} C_VEL
LIN {X 0,Y 126.687,Z 1278.461,A -85,B 0,C 180,E1 23276.488,E2 23276.488} C_VEL
LIN {X 0,Y 119.783,Z 1286.293,A -85,B 0,C 180,E1 23292.492,E2 23292.492} C_VEL
LIN {X 0,Y 118.622,Z 1288.635,A -85,B 0,C 180,E1 23302.705,E2 23302.705} C_VEL
LIN {X 0,Y 119.043,Z 1289.237,A -85,B 0,C 180,E1 23310.014,E2 23310.014} C_VEL
LIN {X 0,Y 119.327,Z 1287.134,A -85,B 0,C 180,E1 23324.665,E2 23324.665} C_VEL
LIN {X 0,Y 125.513,Z 1279.794,A -85,B 0,C 180,E1 23341.476,E2 23341.476} C_VEL
LIN {X 0,Y 140.574,Z 1266.251,A -85,B 0,C 180,E1 23356.739,E2 23356.739} C_VEL
LIN {X 0,Y 155.007,Z 1253.289,A -85,B 0,C 180,E1 23365.064,E2 23365.064} C_VEL
LIN {X 0,Y 154.995,Z 1252.362,A -85,B 0,C 180,E1 23365.958,E2 23365.958} C_VEL
LIN {X 0,Y 131.323,Z 1245.78,A -85,B 0,C 180,E1 23393.401,E2 23393.401} C_VEL
LIN {X 0,Y 155.991,Z 1235.216,A -85,B 0,C 180,E1 23428.924,E2 23428.924} C_VEL
LIN {X 0,Y 168.412,Z 1232.245,A -85,B 0,C 180,E1 23434.459,E2 23434.459} C_VEL
LIN {X 0,Y 150.252,Z 1247.897,A -85,B 0,C 180,E1 23443.252,E2 23443.252} C_VEL
LIN {X 0,Y 133.464,Z 1260.424,A -85,B 0,C 180,E1 23455.559,E2 23455.559} C_VEL
LIN {X 0,Y 122.397,Z 1268.466,A -85,B 0,C 180,E1 23472.033,E2 23472.033} C_VEL
LIN {X 0,Y 119.644,Z 1270.613,A -85,B 0,C 180,E1 23482.74,E2 23482.74} C_VEL
LIN {X 0,Y 119.655,Z 1270.591,A -85,B 0,C 180,E1 23497.231,E2 23497.231} C_VEL
LIN {X 0,Y 125.808,Z 1265.918,A -85,B 0,C 180,E1 23514.666,E2 23514.666} C_VEL
LIN {X 0,Y 132.451,Z 1261.081,A -85,B 0,C 180,E1 23523.354,E2 23523.354} C_VEL
LIN {X 0,Y 136.103,Z 1256.597,A -85,B 0,C 180,E1 23530.426,E2 23530.426} C_VEL
LIN {X 0,Y 141.319,Z 1251.039,A -85,B 0,C 180,E1 23536.957,E2 23536.957} C_VEL
LIN {X 0,Y 163.702,Z 1233.291,A -85,B 0,C 180,E1 23547.245,E2 23547.245} C_VEL
LIN {X 0,Y 188.018,Z 1209.908,A -85,B 0,C 180,E1 23554.527,E2 23554.527} C_VEL
LIN {X 0,Y 210.481,Z 1182.34,A -85,B 0,C 180,E1 23559.453,E2 23559.453} C_VEL
LIN {X 0,Y 224.568,Z 1160.427,A -85,B 0,C 180,E1 23562.205,E2 23562.205} C_VEL
LIN {X 0,Y 226.516,Z 1150.328,A -85,B 0,C 180,E1 23567.497,E2 23567.497} C_VEL
LIN {X 0,Y 227.799,Z 1142.85,A -85,B 0,C 180,E1 23573.486,E2 23573.486} C_VEL
LIN {X 0,Y 228.369,Z 1140.712,A -85,B 0,C 180,E1 23576.212,E2 23576.212} C_VEL
LIN {X 0,Y 228.889,Z 1139.809,A -85,B 0,C 180,E1 23580.001,E2 23580.001} C_VEL
LIN {X 0,Y 229.099,Z 1143.215,A -85,B 0,C 180,E1 23585.591,E2 23585.591} C_VEL
LIN {X 0,Y 229.142,Z 1147.44,A -85,B 0,C 180,E1 23588.987,E2 23588.987} C_VEL
LIN {X 0,Y 223.743,Z 1163.055,A -85,B 0,C 180,E1 23593.143,E2 23593.143} C_VEL
LIN {X 0,Y 203.434,Z 1194.864,A -85,B 0,C 180,E1 23596.585,E2 23596.585} C_VEL
LIN {X 0,Y 180.686,Z 1222.722,A -85,B 0,C 180,E1 23601.724,E2 23601.724} C_VEL
LIN {X 0,Y 158.309,Z 1245.219,A -85,B 0,C 180,E1 23608.841,E2 23608.841} C_VEL
LIN {X 0,Y 136.666,Z 1263.958,A -85,B 0,C 180,E1 23619.401,E2 23619.401} C_VEL
LIN {X 0,Y 119.916,Z 1277.833,A -85,B 0,C 180,E1 23634.318,E2 23634.318} C_VEL
LIN {X 0,Y 112.361,Z 1285.274,A -85,B 0,C 180,E1 23650.065,E2 23650.065} C_VEL
LIN {X 0,Y 110.719,Z 1288.026,A -85,B 0,C 180,E1 23662.182,E2 23662.182} C_VEL
LIN {X 0,Y 111.132,Z 1288.633,A -85,B 0,C 180,E1 23670.015,E2 23670.015} C_VEL
LIN {X 0,Y 111.57,Z 1286.521,A -85,B 0,C 180,E1 23685.71,E2 23685.71} C_VEL
LIN {X 0,Y 118.469,Z 1279.3,A -85,B 0,C 180,E1 23703.315,E2 23703.315} C_VEL
LIN {X 0,Y 135.041,Z 1265.644,A -85,B 0,C 180,E1 23719.27,E2 23719.27} C_VEL
LIN {X 0,Y 146.245,Z 1256.325,A -85,B 0,C 180,E1 23725.659,E2 23725.659} C_VEL
LIN {X 0,Y 134.913,Z 1243.125,A -85,B 0,C 180,E1 23779.604,E2 23779.604} C_VEL
LIN {X 0,Y 158.292,Z 1237.509,A -85,B 0,C 180,E1 23794.027,E2 23794.027} C_VEL
LIN {X 0,Y 156.351,Z 1239.611,A -85,B 0,C 180,E1 23795.561,E2 23795.561} C_VEL
LIN {X 0,Y 134.203,Z 1256.184,A -85,B 0,C 180,E1 23807.554,E2 23807.554} C_VEL
LIN {X 0,Y 119.815,Z 1265.82,A -85,B 0,C 180,E1 23821.83,E2 23821.83} C_VEL
LIN {X 0,Y 113.587,Z 1269.98,A -85,B 0,C 180,E1 23834.576,E2 23834.576} C_VEL
LIN {X 0,Y 111.391,Z 1271.65,A -85,B 0,C 180,E1 23849.985,E2 23849.985} C_VEL
LIN {X 0,Y 113.579,Z 1269.945,A -85,B 0,C 180,E1 23865.395,E2 23865.395} C_VEL
LIN {X 0,Y 123.868,Z 1263.076,A -85,B 0,C 180,E1 23883.229,E2 23883.229} C_VEL
LIN {X 0,Y 141.319,Z 1251.039,A -85,B 0,C 180,E1 23896.957,E2 23896.957} C_VEL
LIN {X 0,Y 147.8,Z 1244.617,A -85,B 0,C 180,E1 23902.882,E2 23902.882} C_VEL
LIN {X 0,Y 155.408,Z 1237.312,A -85,B 0,C 180,E1 23908.189,E2 23908.189} C_VEL
LIN {X 0,Y 179.936,Z 1215.346,A -85,B 0,C 180,E1 23915.602,E2 23915.602} C_VEL
LIN {X 0,Y 203.674,Z 1188.458,A -85,B 0,C 180,E1 23920.736,E2 23920.736} C_VEL
LIN {X 0,Y 220.178,Z 1164.682,A -85,B 0,C 180,E1 23923.617,E2 23923.617} C_VEL
LIN {X 0,Y 222.596,Z 1154.834,A -85,B 0,C 180,E1 23929.257,E2 23929.257} C_VEL
LIN {X 0,Y 224.139,Z 1148.821,A -85,B 0,C 180,E1 23934.762,E2 23934.762} C_VEL
LIN {X 0,Y 225.174,Z 1146.834,A -85,B 0,C 180,E1 23940.001,E2 23940.001} C_VEL
LIN {X 0,Y 225.225,Z 1150.383,A -85,B 0,C 180,E1 23945.688,E2 23945.688} C_VEL
LIN {X 0,Y 224.925,Z 1153.606,A -85,B 0,C 180,E1 23948.072,E2 23948.072} C_VEL
LIN {X 0,Y 219.755,Z 1166.545,A -85,B 0,C 180,E1 23951.456,E2 23951.456} C_VEL
LIN {X 0,Y 197.775,Z 1198.776,A -85,B 0,C 180,E1 23955.006,E2 23955.006} C_VEL
LIN {X 0,Y 173.506,Z 1226.587,A -85,B 0,C 180,E1 23960.358,E2 23960.358} C_VEL
LIN {X 0,Y 148.141,Z 1250.067,A -85,B 0,C 180,E1 23968.55,E2 23968.55} C_VEL
LIN {X 0,Y 125.671,Z 1267.804,A -85,B 0,C 180,E1 23980.443,E2 23980.443} C_VEL
LIN {X 0,Y 109.96,Z 1279.915,A -85,B 0,C 180,E1 23996.723,E2 23996.723} C_VEL
LIN {X 0,Y 103.771,Z 1285.886,A -85,B 0,C 180,E1 24013.108,E2 24013.108} C_VEL
LIN {X 0,Y 103.238,Z 1288.031,A -85,B 0,C 180,E1 24030.016,E2 24030.016} C_VEL
LIN {X 0,Y 103.834,Z 1285.906,A -85,B 0,C 180,E1 24046.915,E2 24046.915} C_VEL
LIN {X 0,Y 112.087,Z 1278.4,A -85,B 0,C 180,E1 24066.122,E2 24066.122} C_VEL
LIN {X 0,Y 130.122,Z 1264.766,A -85,B 0,C 180,E1 24082.229,E2 24082.229} C_VEL
LIN {X 0,Y 137.079,Z 1259.022,A -85,B 0,C 180,E1 24086.605,E2 24086.605} C_VEL
LIN {X 0,Y 117.495,Z 1251.738,A -85,B 0,C 180,E1 24119.999,E2 24119.999} C_VEL
LIN {X 0,Y 148.338,Z 1242.377,A -85,B 0,C 180,E1 24153.636,E2 24153.636} C_VEL
LIN {X 0,Y 147.33,Z 1243.67,A -85,B 0,C 180,E1 24154.954,E2 24154.954} C_VEL
LIN {X 0,Y 126.356,Z 1258.059,A -85,B 0,C 180,E1 24166.611,E2 24166.611} C_VEL
LIN {X 0,Y 112.234,Z 1266.781,A -85,B 0,C 180,E1 24180.821,E2 24180.821} C_VEL
LIN {X 0,Y 105.961,Z 1270.585,A -85,B 0,C 180,E1 24193.435,E2 24193.435} C_VEL
LIN {X 0,Y 103.532,Z 1272.25,A -85,B 0,C 180,E1 24209.984,E2 24209.984} C_VEL
LIN {X 0,Y 105.954,Z 1270.55,A -85,B 0,C 180,E1 24226.533,E2 24226.533} C_VEL
LIN {X 0,Y 117.276,Z 1263.685,A -85,B 0,C 180,E1 24245.366,E2 24245.366} C_VEL
LIN {X 0,Y 137.427,Z 1250.631,A -85,B 0,C 180,E1 24260.214,E2 24260.214} C_VEL
LIN {X 0,Y 155.408,Z 1237.312,A -85,B 0,C 180,E1 24268.189,E2 24268.189} C_VEL
LIN {X 0,Y 163.814,Z 1229.081,A -85,B 0,C 180,E1 24272.874,E2 24272.874} C_VEL
LIN {X 0,Y 172.711,Z 1219.867,A -85,B 0,C 180,E1 24276.951,E2 24276.951} C_VEL
LIN {X 0,Y 197.4,Z 1193.736,A -85,B 0,C 180,E1 24282.197,E2 24282.197} C_VEL
LIN {X 0,Y 215.698,Z 1169.073,A -85,B 0,C 180,E1 24285.243,E2 24285.243} C_VEL
LIN {X 0,Y 217.986,Z 1162.22,A -85,B 0,C 180,E1 24289.011,E2 24289.011} C_VEL
LIN {X 0,Y 219.8,Z 1156.347,A -85,B 0,C 180,E1 24294.09,E2 24294.09} C_VEL
LIN {X 0,Y 221.276,Z 1153.77,A -85,B 0,C 180,E1 24300.001,E2 24300.001} C_VEL
LIN {X 0,Y 221.141,Z 1157.566,A -85,B 0,C 180,E1 24305.875,E2 24305.875} C_VEL
LIN {X 0,Y 221.03,Z 1158.705,A -85,B 0,C 180,E1 24306.862,E2 24306.862} C_VEL
LIN {X 0,Y 216.176,Z 1169.342,A -85,B 0,C 180,E1 24309.662,E2 24309.662} C_VEL
LIN {X 0,Y 194.481,Z 1199.836,A -85,B 0,C 180,E1 24312.938,E2 24312.938} C_VEL
LIN {X 0,Y 168.759,Z 1228.028,A -85,B 0,C 180,E1 24318.288,E2 24318.288} C_VEL
LIN {X 0,Y 142.951,Z 1250.561,A -85,B 0,C 180,E1 24326.221,E2 24326.221} C_VEL
LIN {X 0,Y 119.672,Z 1267.754,A -85,B 0,C 180,E1 24338.013,E2 24338.013} C_VEL
LIN {X 0,Y 103.219,Z 1279.291,A -85,B 0,C 180,E1 24354.231,E2 24354.231} C_VEL
LIN {X 0,Y 96.073,Z 1285.27,A -85,B 0,C 180,E1 24371.709,E2 24371.709} C_VEL
LIN {X 0,Y 95.319,Z 1287.426,A -85,B 0,C 180,E1 24390.017,E2 24390.017} C_VEL
LIN {X 0,Y 96.595,Z 1284.844,A -85,B 0,C 180,E1 24410.396,E2 24410.396} C_VEL
LIN {X 0,Y 107.572,Z 1276.386,A -85,B 0,C 180,E1 24431.145,E2 24431.145} C_VEL
LIN {X 0,Y 127.072,Z 1262.793,A -85,B 0,C 180,E1 24446.255,E2 24446.255} C_VEL
LIN {X 0,Y 123.343,Z 1261.148,A -85,B 0,C 180,E1 24450.701,E2 24450.701} C_VEL
LIN {X 0,Y 129.265,Z 1248.791,A -85,B 0,C 180,E1 24507.834,E2 24507.834} C_VEL
LIN {X 0,Y 138.959,Z 1246.778,A -85,B 0,C 180,E1 24513.552,E2 24513.552} C_VEL
LIN {X 0,Y 120.684,Z 1258.666,A -85,B 0,C 180,E1 24524.009,E2 24524.009} C_VEL
LIN {X 0,Y 104.233,Z 1267.979,A -85,B 0,C 180,E1 24540.293,E2 24540.293} C_VEL
LIN {X 0,Y 96.19,Z 1272.421,A -85,B 0,C 180,E1 24560.956,E2 24560.956} C_VEL
LIN {X 0,Y 96.196,Z 1272.399,A -85,B 0,C 180,E1 24579.008,E2 24579.008} C_VEL
LIN {X 0,Y 104.494,Z 1267.802,A -85,B 0,C 180,E1 24599.957,E2 24599.957} C_VEL
LIN {X 0,Y 122.923,Z 1257.292,A -85,B 0,C 180,E1 24617.421,E2 24617.421} C_VEL
LIN {X 0,Y 147.432,Z 1240.819,A -85,B 0,C 180,E1 24629.354,E2 24629.354} C_VEL
LIN {X 0,Y 172.711,Z 1219.867,A -85,B 0,C 180,E1 24636.951,E2 24636.951} C_VEL
LIN {X 0,Y 181.897,Z 1209.893,A -85,B 0,C 180,E1 24640.555,E2 24640.555} C_VEL
LIN {X 0,Y 189.695,Z 1200.52,A -85,B 0,C 180,E1 24643.444,E2 24643.444} C_VEL
LIN {X 0,Y 191.029,Z 1199.011,A -85,B 0,C 180,E1 24643.711,E2 24643.711} C_VEL
LIN {X 0,Y 211.977,Z 1172.269,A -85,B 0,C 180,E1 24647.077,E2 24647.077} C_VEL
LIN {X 0,Y 214.989,Z 1164.225,A -85,B 0,C 180,E1 24653.066,E2 24653.066} C_VEL
LIN {X 0,Y 216.14,Z 1161.768,A -85,B 0,C 180,E1 24655.998,E2 24655.998} C_VEL
LIN {X 0,Y 217.093,Z 1160.517,A -85,B 0,C 180,E1 24660.001,E2 24660.001} C_VEL
LIN {X 0,Y 216.72,Z 1164.556,A -85,B 0,C 180,E1 24665.815,E2 24665.815} C_VEL
LIN {X 0,Y 212.366,Z 1172.791,A -85,B 0,C 180,E1 24667.858,E2 24667.858} C_VEL
LIN {X 0,Y 188.928,Z 1203.878,A -85,B 0,C 180,E1 24671.215,E2 24671.215} C_VEL
LIN {X 0,Y 162.764,Z 1230.664,A -85,B 0,C 180,E1 24676.438,E2 24676.438} C_VEL
LIN {X 0,Y 135.057,Z 1253.297,A -85,B 0,C 180,E1 24684.82,E2 24684.82} C_VEL
LIN {X 0,Y 110.685,Z 1269.764,A -85,B 0,C 180,E1 24697.546,E2 24697.546} C_VEL
LIN {X 0,Y 93.869,Z 1280.516,A -85,B 0,C 180,E1 24715.781,E2 24715.781} C_VEL
LIN {X 0,Y 88.471,Z 1284.656,A -85,B 0,C 180,E1 24730.074,E2 24730.074} C_VEL
LIN {X 0,Y 87.401,Z 1286.822,A -85,B 0,C 180,E1 24750.019,E2 24750.019} C_VEL
LIN {X 0,Y 88.537,Z 1284.677,A -85,B 0,C 180,E1 24769.951,E2 24769.951} C_VEL
LIN {X 0,Y 100.16,Z 1276.64,A -85,B 0,C 180,E1 24792.704,E2 24792.704} C_VEL
LIN {X 0,Y 115.703,Z 1266.778,A -85,B 0,C 180,E1 24805.509,E2 24805.509} C_VEL
LIN {X 0,Y 117.883,Z 1264.844,A -85,B 0,C 180,E1 24807.729,E2 24807.729} C_VEL
LIN {X 0,Y 128.976,Z 1250.996,A -85,B 0,C 180,E1 24873.091,E2 24873.091} C_VEL
LIN {X 0,Y 116.598,Z 1258.566,A -85,B 0,C 180,E1 24880.319,E2 24880.319} C_VEL
LIN {X 0,Y 97.399,Z 1268.586,A -85,B 0,C 180,E1 24897.971,E2 24897.971} C_VEL
LIN {X 0,Y 88.417,Z 1273.022,A -85,B 0,C 180,E1 24920.154,E2 24920.154} C_VEL
LIN {X 0,Y 88.42,Z 1273.001,A -85,B 0,C 180,E1 24939.808,E2 24939.808} C_VEL
LIN {X 0,Y 97.694,Z 1268.408,A -85,B 0,C 180,E1 24962.283,E2 24962.283} C_VEL
LIN {X 0,Y 117.667,Z 1257.902,A -85,B 0,C 180,E1 24980.285,E2 24980.285} C_VEL
LIN {X 0,Y 142.555,Z 1242.128,A -85,B 0,C 180,E1 24991.746,E2 24991.746} C_VEL
LIN {X 0,Y 169.041,Z 1221.103,A -85,B 0,C 180,E1 24999.25,E2 24999.25} C_VEL
LIN {X 0,Y 191.029,Z 1199.011,A -85,B 0,C 180,E1 25003.711,E2 25003.711} C_VEL
LIN {X 0,Y 196.623,Z 1191.706,A -85,B 0,C 180,E1 25005.912,E2 25005.912} C_VEL
LIN {X 0,Y 202.072,Z 1184.063,A -85,B 0,C 180,E1 25008,E2 25008} C_VEL
LIN {X 0,Y 207.364,Z 1177.066,A -85,B 0,C 180,E1 25008.748,E2 25008.748} C_VEL
LIN {X 0,Y 209.65,Z 1172.428,A -85,B 0,C 180,E1 25011.724,E2 25011.724} C_VEL
LIN {X 0,Y 211.695,Z 1168.302,A -85,B 0,C 180,E1 25016.234,E2 25016.234} C_VEL
LIN {X 0,Y 212.735,Z 1167.166,A -85,B 0,C 180,E1 25020.001,E2 25020.001} C_VEL
LIN {X 0,Y 212.01,Z 1170.704,A -85,B 0,C 180,E1 25024.891,E2 25024.891} C_VEL
LIN {X 0,Y 209.377,Z 1175.269,A -85,B 0,C 180,E1 25025.916,E2 25025.916} C_VEL
LIN {X 0,Y 185.286,Z 1205.715,A -85,B 0,C 180,E1 25029.12,E2 25029.12} C_VEL
LIN {X 0,Y 158.92,Z 1231.555,A -85,B 0,C 180,E1 25034.007,E2 25034.007} C_VEL
LIN {X 0,Y 130.274,Z 1253.701,A -85,B 0,C 180,E1 25042.108,E2 25042.108} C_VEL
LIN {X 0,Y 105.27,Z 1269.477,A -85,B 0,C 180,E1 25054.412,E2 25054.412} C_VEL
LIN {X 0,Y 87.112,Z 1279.964,A -85,B 0,C 180,E1 25072.963,E2 25072.963} C_VEL
LIN {X 0,Y 80.674,Z 1284.246,A -85,B 0,C 180,E1 25089.267,E2 25089.267} C_VEL
LIN {X 0,Y 79.476,Z 1286.217,A -85,B 0,C 180,E1 25110.021,E2 25110.021} C_VEL
LIN {X 0,Y 81.004,Z 1284.062,A -85,B 0,C 180,E1 25131.897,E2 25131.897} C_VEL
LIN {X 0,Y 94.32,Z 1276.016,A -85,B 0,C 180,E1 25156.077,E2 25156.077} C_VEL
LIN {X 0,Y 107.956,Z 1268.179,A -85,B 0,C 180,E1 25167.032,E2 25167.032} C_VEL
LIN {X 0,Y 109.058,Z 1267.113,A -85,B 0,C 180,E1 25168.451,E2 25168.451} C_VEL
LIN {X 0,Y 118.43,Z 1255.076,A -85,B 0,C 180,E1 25232.284,E2 25232.284} C_VEL
LIN {X 0,Y 115.948,Z 1256.829,A -85,B 0,C 180,E1 25234.79,E2 25234.79} C_VEL
LIN {X 0,Y 94.828,Z 1267.379,A -85,B 0,C 180,E1 25250.442,E2 25250.442} C_VEL
LIN {X 0,Y 83.462,Z 1272.397,A -85,B 0,C 180,E1 25268.779,E2 25268.779} C_VEL
LIN {X 0,Y 79.903,Z 1274.053,A -85,B 0,C 180,E1 25289.979,E2 25289.979} C_VEL
LIN {X 0,Y 83.456,Z 1272.364,A -85,B 0,C 180,E1 25311.18,E2 25311.18} C_VEL
LIN {X 0,Y 98.746,Z 1265.511,A -85,B 0,C 180,E1 25333.425,E2 25333.425} C_VEL
LIN {X 0,Y 123.485,Z 1252.458,A -85,B 0,C 180,E1 25348.782,E2 25348.782} C_VEL
LIN {X 0,Y 150.487,Z 1234.557,A -85,B 0,C 180,E1 25358.03,E2 25358.03} C_VEL
LIN {X 0,Y 178.389,Z 1210.626,A -85,B 0,C 180,E1 25364.172,E2 25364.172} C_VEL
LIN {X 0,Y 202.072,Z 1184.063,A -85,B 0,C 180,E1 25368,E2 25368} C_VEL
LIN {X 0,Y 204.757,Z 1180.039,A -85,B 0,C 180,E1 25369.402,E2 25369.402} C_VEL
LIN {X 0,Y 205.934,Z 1176.554,A -85,B 0,C 180,E1 25374.222,E2 25374.222} C_VEL
LIN {X 0,Y 208.219,Z 1173.702,A -85,B 0,C 180,E1 25380.001,E2 25380.001} C_VEL
LIN {X 0,Y 207.769,Z 1175.85,A -85,B 0,C 180,E1 25383.645,E2 25383.645} C_VEL
LIN {X 0,Y 184.164,Z 1205.094,A -85,B 0,C 180,E1 25386.599,E2 25386.599} C_VEL
LIN {X 0,Y 156.335,Z 1231.618,A -85,B 0,C 180,E1 25391.262,E2 25391.262} C_VEL
LIN {X 0,Y 127.406,Z 1253.074,A -85,B 0,C 180,E1 25398.679,E2 25398.679} C_VEL
LIN {X 0,Y 101.134,Z 1268.689,A -85,B 0,C 180,E1 25410.358,E2 25410.358} C_VEL
LIN {X 0,Y 79.955,Z 1279.752,A -85,B 0,C 180,E1 25430.691,E2 25430.691} C_VEL
LIN {X 0,Y 73.456,Z 1283.419,A -85,B 0,C 180,E1 25445.765,E2 25445.765} C_VEL
LIN {X 0,Y 71.546,Z 1285.612,A -85,B 0,C 180,E1 25470.023,E2 25470.023} C_VEL
LIN {X 0,Y 73.554,Z 1283.445,A -85,B 0,C 180,E1 25494.25,E2 25494.25} C_VEL
LIN {X 0,Y 88.81,Z 1275.39,A -85,B 0,C 180,E1 25519.904,E2 25519.904} C_VEL
LIN {X 0,Y 100.186,Z 1269.366,A -85,B 0,C 180,E1 25528.824,E2 25528.824} C_VEL
LIN {X 0,Y 108.664,Z 1258.686,A -85,B 0,C 180,E1 25591.89,E2 25591.89} C_VEL
LIN {X 0,Y 108.171,Z 1259.216,A -85,B 0,C 180,E1 25593.143,E2 25593.143} C_VEL
LIN {X 0,Y 84.893,Z 1269.57,A -85,B 0,C 180,E1 25611.501,E2 25611.501} C_VEL
LIN {X 0,Y 76.121,Z 1273.002,A -85,B 0,C 180,E1 25626.617,E2 25626.617} C_VEL
LIN {X 0,Y 72.045,Z 1274.653,A -85,B 0,C 180,E1 25649.977,E2 25649.977} C_VEL
LIN {X 0,Y 78.499,Z 1272.056,A -85,B 0,C 180,E1 25678.649,E2 25678.649} C_VEL
LIN {X 0,Y 97.798,Z 1263.989,A -85,B 0,C 180,E1 25700.463,E2 25700.463} C_VEL
LIN {X 0,Y 125.31,Z 1249.816,A -85,B 0,C 180,E1 25714.262,E2 25714.262} C_VEL
LIN {X 0,Y 152.651,Z 1231.483,A -85,B 0,C 180,E1 25722.046,E2 25722.046} C_VEL
LIN {X 0,Y 179.847,Z 1207.831,A -85,B 0,C 180,E1 25727.229,E2 25727.229} C_VEL
LIN {X 0,Y 203.21,Z 1181.337,A -85,B 0,C 180,E1 25730.562,E2 25730.562} C_VEL
LIN {X 0,Y 205.106,Z 1178.097,A -85,B 0,C 180,E1 25732.604,E2 25732.604} C_VEL
LIN {X 0,Y 205.934,Z 1176.554,A -85,B 0,C 180,E1 25734.222,E2 25734.222} C_VEL
LIN {X 0,Y 205.569,Z 1176.773,A -85,B 0,C 180,E1 25736.64,E2 25736.64} C_VEL
LIN {X 0,Y 203.306,Z 1180.429,A -85,B 0,C 180,E1 25740.731,E2 25740.731} C_VEL
LIN {X 0,Y 202.817,Z 1181.56,A -85,B 0,C 180,E1 25742.012,E2 25742.012} C_VEL
LIN {X 0,Y 177.07,Z 1211.045,A -85,B 0,C 180,E1 25744.889,E2 25744.889} C_VEL
LIN {X 0,Y 149.098,Z 1235.6,A -85,B 0,C 180,E1 25749.381,E2 25749.381} C_VEL
LIN {X 0,Y 118.424,Z 1256.492,A -85,B 0,C 180,E1 25757.163,E2 25757.163} C_VEL
LIN {X 0,Y 91.444,Z 1270.979,A -85,B 0,C 180,E1 25769.674,E2 25769.674} C_VEL
LIN {X 0,Y 71.31,Z 1280.315,A -85,B 0,C 180,E1 25790.621,E2 25790.621} C_VEL
LIN {X 0,Y 63.571,Z 1284.368,A -85,B 0,C 180,E1 25816.295,E2 25816.295} C_VEL
LIN {X 0,Y 63.614,Z 1285.007,A -85,B 0,C 180,E1 25830.026,E2 25830.026} C_VEL
LIN {X 0,Y 66.261,Z 1282.828,A -85,B 0,C 180,E1 25857.124,E2 25857.124} C_VEL
LIN {X 0,Y 83.768,Z 1274.766,A -85,B 0,C 180,E1 25884.194,E2 25884.194} C_VEL
LIN {X 0,Y 90.604,Z 1271.339,A -85,B 0,C 180,E1 25890.023,E2 25890.023} C_VEL
LIN {X 0,Y 98.695,Z 1262.019,A -85,B 0,C 180,E1 25951.344,E2 25951.344} C_VEL
LIN {X 0,Y 96.031,Z 1263.423,A -85,B 0,C 180,E1 25953.78,E2 25953.78} C_VEL
LIN {X 0,Y 73.291,Z 1272.132,A -85,B 0,C 180,E1 25975.436,E2 25975.436} C_VEL
LIN {X 0,Y 65.175,Z 1274.831,A -85,B 0,C 180,E1 25996.586,E2 25996.586} C_VEL
LIN {X 0,Y 64.16,Z 1275.255,A -85,B 0,C 180,E1 26009.974,E2 26009.974} C_VEL
LIN {X 0,Y 68.918,Z 1273.574,A -85,B 0,C 180,E1 26035.945,E2 26035.945} C_VEL
LIN {X 0,Y 87.856,Z 1266.728,A -85,B 0,C 180,E1 26060.589,E2 26060.589} C_VEL
LIN {X 0,Y 116.021,Z 1253.675,A -85,B 0,C 180,E1 26075.536,E2 26075.536} C_VEL
LIN {X 0,Y 145.284,Z 1235.769,A -85,B 0,C 180,E1 26083.861,E2 26083.861} C_VEL
LIN {X 0,Y 174.729,Z 1211.83,A -85,B 0,C 180,E1 26089.186,E2 26089.186} C_VEL
LIN {X 0,Y 199.135,Z 1185.565,A -85,B 0,C 180,E1 26092.428,E2 26092.428} C_VEL
LIN {X 0,Y 201.205,Z 1182.572,A -85,B 0,C 180,E1 26094.826,E2 26094.826} C_VEL
LIN {X 0,Y 203.306,Z 1180.429,A -85,B 0,C 180,E1 26100.731,E2 26100.731} C_VEL
LIN {X 0,Y 201.17,Z 1183.49,A -85,B 0,C 180,E1 26101.544,E2 26101.544} C_VEL
LIN {X 0,Y 188.013,Z 1198.51,A -85,B 0,C 180,E1 26101.002,E2 26101.002} C_VEL
LIN {X 0,Y 158.912,Z 1226.34,A -85,B 0,C 180,E1 26104.501,E2 26104.501} C_VEL
LIN {X 0,Y 128.481,Z 1248.471,A -85,B 0,C 180,E1 26110.117,E2 26110.117} C_VEL
LIN {X 0,Y 96.579,Z 1266.211,A -85,B 0,C 180,E1 26120.412,E2 26120.412} C_VEL
LIN {X 0,Y 70.805,Z 1277.426,A -85,B 0,C 180,E1 26138.547,E2 26138.547} C_VEL
LIN {X 0,Y 59.042,Z 1282.181,A -85,B 0,C 180,E1 26159.291,E2 26159.291} C_VEL
LIN {X 0,Y 55.68,Z 1284.401,A -85,B 0,C 180,E1 26190.03,E2 26190.03} C_VEL
LIN {X 0,Y 59.155,Z 1282.209,A -85,B 0,C 180,E1 26220.71,E2 26220.71} C_VEL
LIN {X 0,Y 79.231,Z 1274.138,A -85,B 0,C 180,E1 26249.032,E2 26249.032} C_VEL
LIN {X 0,Y 80.626,Z 1272.948,A -85,B 0,C 180,E1 26252.101,E2 26252.101} C_VEL
LIN {X 0,Y 88.701,Z 1265.114,A -85,B 0,C 180,E1 26310.685,E2 26310.685} C_VEL
LIN {X 0,Y 73.12,Z 1270.782,A -85,B 0,C 180,E1 26323.72,E2 26323.72} C_VEL
LIN {X 0,Y 57.521,Z 1275.434,A -85,B 0,C 180,E1 26354.761,E2 26354.761} C_VEL
LIN {X 0,Y 56.275,Z 1275.857,A -85,B 0,C 180,E1 26369.97,E2 26369.97} C_VEL
LIN {X 0,Y 61.892,Z 1274.179,A -85,B 0,C 180,E1 26399.155,E2 26399.155} C_VEL
LIN {X 0,Y 83.018,Z 1267.337,A -85,B 0,C 180,E1 26424.849,E2 26424.849} C_VEL
LIN {X 0,Y 112.946,Z 1254.285,A -85,B 0,C 180,E1 26439.228,E2 26439.228} C_VEL
LIN {X 0,Y 144.497,Z 1235.562,A -85,B 0,C 180,E1 26447.156,E2 26447.156} C_VEL
LIN {X 0,Y 173.027,Z 1212.798,A -85,B 0,C 180,E1 26451.716,E2 26451.716} C_VEL
LIN {X 0,Y 195.396,Z 1189.652,A -85,B 0,C 180,E1 26454.373,E2 26454.373} C_VEL
LIN {X 0,Y 196.643,Z 1188.003,A -85,B 0,C 180,E1 26455.933,E2 26455.933} C_VEL
LIN {X 0,Y 198.387,Z 1186.353,A -85,B 0,C 180,E1 26460.001,E2 26460.001} C_VEL
LIN {X 0,Y 188.013,Z 1198.51,A -85,B 0,C 180,E1 26461.002,E2 26461.002} C_VEL
LIN {X 0,Y 175.592,Z 1210.926,A -85,B 0,C 180,E1 26461.003,E2 26461.003} C_VEL
LIN {X 0,Y 162.421,Z 1222.47,A -85,B 0,C 180,E1 26461.099,E2 26461.099} C_VEL
LIN {X 0,Y 130.096,Z 1246.101,A -85,B 0,C 180,E1 26465.898,E2 26465.898} C_VEL
LIN {X 0,Y 98.724,Z 1263.337,A -85,B 0,C 180,E1 26473.969,E2 26473.969} C_VEL
LIN {X 0,Y 69.487,Z 1275.528,A -85,B 0,C 180,E1 26489.742,E2 26489.742} C_VEL
LIN {X 0,Y 52.238,Z 1281.562,A -85,B 0,C 180,E1 26514.746,E2 26514.746} C_VEL
LIN {X 0,Y 47.737,Z 1283.795,A -85,B 0,C 180,E1 26550.035,E2 26550.035} C_VEL
LIN {X 0,Y 52.345,Z 1281.59,A -85,B 0,C 180,E1 26585.25,E2 26585.25} C_VEL
LIN {X 0,Y 69.669,Z 1275.592,A -85,B 0,C 180,E1 26610.092,E2 26610.092} C_VEL
LIN {X 0,Y 71.623,Z 1274.543,A -85,B 0,C 180,E1 26613.051,E2 26613.051} C_VEL
LIN {X 0,Y 78.192,Z 1268.052,A -85,B 0,C 180,E1 26669.246,E2 26669.246} C_VEL
LIN {X 0,Y 73.131,Z 1269.806,A -85,B 0,C 180,E1 26674.331,E2 26674.331} C_VEL
LIN {X 0,Y 55.11,Z 1274.815,A -85,B 0,C 180,E1 26696.758,E2 26696.758} C_VEL
LIN {X 0,Y 48.389,Z 1276.458,A -85,B 0,C 180,E1 26729.966,E2 26729.966} C_VEL
LIN {X 0,Y 58.121,Z 1274.047,A -85,B 0,C 180,E1 26768.848,E2 26768.848} C_VEL
LIN {X 0,Y 84.62,Z 1265.813,A -85,B 0,C 180,E1 26793.039,E2 26793.039} C_VEL
LIN {X 0,Y 116.718,Z 1251.753,A -85,B 0,C 180,E1 26804.826,E2 26804.826} C_VEL
LIN {X 0,Y 146.469,Z 1233.72,A -85,B 0,C 180,E1 26810.828,E2 26810.828} C_VEL
LIN {X 0,Y 175.491,Z 1210.22,A -85,B 0,C 180,E1 26814.734,E2 26814.734} C_VEL
LIN {X 0,Y 190.238,Z 1195.285,A -85,B 0,C 180,E1 26816.257,E2 26816.257} C_VEL
LIN {X 0,Y 191.736,Z 1193.652,A -85,B 0,C 180,E1 26816.907,E2 26816.907} C_VEL
LIN {X 0,Y 192.075,Z 1193.346,A -85,B 0,C 180,E1 26817.747,E2 26817.747} C_VEL
LIN {X 0,Y 189.899,Z 1195.829,A -85,B 0,C 180,E1 26818.384,E2 26818.384} C_VEL
LIN {X 0,Y 162.421,Z 1222.47,A -85,B 0,C 180,E1 26821.099,E2 26821.099} C_VEL
LIN {X 0,Y 148.478,Z 1233.105,A -85,B 0,C 180,E1 26821.294,E2 26821.294} C_VEL
LIN {X 0,Y 133.872,Z 1242.76,A -85,B 0,C 180,E1 26821.625,E2 26821.625} C_VEL
LIN {X 0,Y 102.076,Z 1260.441,A -85,B 0,C 180,E1 26827.87,E2 26827.87} C_VEL
LIN {X 0,Y 71.376,Z 1273.03,A -85,B 0,C 180,E1 26839.877,E2 26839.877} C_VEL
LIN {X 0,Y 45.844,Z 1280.942,A -85,B 0,C 180,E1 26868.874,E2 26868.874} C_VEL
LIN {X 0,Y 39.801,Z 1283.189,A -85,B 0,C 180,E1 26910.042,E2 26910.042} C_VEL
LIN {X 0,Y 45.952,Z 1280.971,A -85,B 0,C 180,E1 26951.105,E2 26951.105} C_VEL
LIN {X 0,Y 61.707,Z 1276.337,A -85,B 0,C 180,E1 26972.94,E2 26972.94} C_VEL
LIN {X 0,Y 61.057,Z 1275.562,A -85,B 0,C 180,E1 26978.238,E2 26978.238} C_VEL
LIN {X 0,Y 68.161,Z 1270.568,A -85,B 0,C 180,E1 27028.092,E2 27028.092} C_VEL
LIN {X 0,Y 63.033,Z 1272.032,A -85,B 0,C 180,E1 27033.355,E2 27033.355} C_VEL
LIN {X 0,Y 48.677,Z 1275.42,A -85,B 0,C 180,E1 27051.638,E2 27051.638} C_VEL
LIN {X 0,Y 40.51,Z 1277.06,A -85,B 0,C 180,E1 27089.959,E2 27089.959} C_VEL
LIN {X 0,Y 52.178,Z 1274.653,A -85,B 0,C 180,E1 27134.322,E2 27134.322} C_VEL
LIN {X 0,Y 81.322,Z 1266.421,A -85,B 0,C 180,E1 27158.044,E2 27158.044} C_VEL
LIN {X 0,Y 114.479,Z 1252.577,A -85,B 0,C 180,E1 27168.567,E2 27168.567} C_VEL
LIN {X 0,Y 146.777,Z 1233.372,A -85,B 0,C 180,E1 27174.1,E2 27174.1} C_VEL
LIN {X 0,Y 173.258,Z 1212.36,A -85,B 0,C 180,E1 27177.16,E2 27177.16} C_VEL
LIN {X 0,Y 143.341,Z 1236.437,A -85,B 0,C 180,E1 27180.326,E2 27180.326} C_VEL
LIN {X 0,Y 133.872,Z 1242.76,A -85,B 0,C 180,E1 27181.625,E2 27181.625} C_VEL
LIN {X 0,Y 118.621,Z 1251.401,A -85,B 0,C 180,E1 27182.117,E2 27182.117} C_VEL
LIN {X 0,Y 102.922,Z 1259.017,A -85,B 0,C 180,E1 27182.885,E2 27182.885} C_VEL
LIN {X 0,Y 67.369,Z 1272.907,A -85,B 0,C 180,E1 27194.257,E2 27194.257} C_VEL
LIN {X 0,Y 40.072,Z 1280.321,A -85,B 0,C 180,E1 27221.198,E2 27221.198} C_VEL
LIN {X 0,Y 31.845,Z 1282.582,A -85,B 0,C 180,E1 27270.052,E2 27270.052} C_VEL
LIN {X 0,Y 40.18,Z 1280.351,A -85,B 0,C 180,E1 27318.752,E2 27318.752} C_VEL
LIN {X 0,Y 52.192,Z 1277.443,A -85,B 0,C 180,E1 27335.08,E2 27335.08} C_VEL
LIN {X 0,Y 52.675,Z 1276.818,A -85,B 0,C 180,E1 27339.06,E2 27339.06} C_VEL
LIN {X 0,Y 57.398,Z 1272.958,A -85,B 0,C 180,E1 27385.229,E2 27385.229} C_VEL
LIN {X 0,Y 57.073,Z 1273.106,A -85,B 0,C 180,E1 27388.356,E2 27388.356} C_VEL
LIN {X 0,Y 35.194,Z 1277.243,A -85,B 0,C 180,E1 27424.557,E2 27424.557} C_VEL
LIN {X 0,Y 32.623,Z 1277.662,A -85,B 0,C 180,E1 27449.949,E2 27449.949} C_VEL
LIN {X 0,Y 43.2,Z 1275.915,A -85,B 0,C 180,E1 27495.693,E2 27495.693} C_VEL
LIN {X 0,Y 71.69,Z 1269.235,A -85,B 0,C 180,E1 27520.493,E2 27520.493} C_VEL
LIN {X 0,Y 103.237,Z 1257.767,A -85,B 0,C 180,E1 27530.535,E2 27530.535} C_VEL
LIN {X 0,Y 136.111,Z 1240.512,A -85,B 0,C 180,E1 27536.04,E2 27536.04} C_VEL
LIN {X 0,Y 143.809,Z 1235.605,A -85,B 0,C 180,E1 27536.935,E2 27536.935} C_VEL
LIN {X 0,Y 109.172,Z 1255.983,A -85,B 0,C 180,E1 27541.706,E2 27541.706} C_VEL
LIN {X 0,Y 102.922,Z 1259.017,A -85,B 0,C 180,E1 27542.885,E2 27542.885} C_VEL
LIN {X 0,Y 86.757,Z 1265.621,A -85,B 0,C 180,E1 27543.968,E2 27543.968} C_VEL
LIN {X 0,Y 70.199,Z 1270.942,A -85,B 0,C 180,E1 27545.687,E2 27545.687} C_VEL
LIN {X 0,Y 44.724,Z 1277.758,A -85,B 0,C 180,E1 27559.722,E2 27559.722} C_VEL
LIN {X 0,Y 26.312,Z 1281.3,A -85,B 0,C 180,E1 27595.082,E2 27595.082} C_VEL
LIN {X 0,Y 23.89,Z 1281.975,A -85,B 0,C 180,E1 27630.07,E2 27630.07} C_VEL
LIN {X 0,Y 35.348,Z 1279.73,A -85,B 0,C 180,E1 27688.72,E2 27688.72} C_VEL
LIN {X 0,Y 44.279,Z 1277.875,A -85,B 0,C 180,E1 27700.072,E2 27700.072} C_VEL
LIN {X 0,Y 47.321,Z 1275.014,A -85,B 0,C 180,E1 27742.265,E2 27742.265} C_VEL
LIN {X 0,Y 46.755,Z 1275.1,A -85,B 0,C 180,E1 27746.01,E2 27746.01} C_VEL
LIN {X 0,Y 28.254,Z 1277.847,A -85,B 0,C 180,E1 27777.647,E2 27777.647} C_VEL
LIN {X 0,Y 24.745,Z 1278.263,A -85,B 0,C 180,E1 27809.933,E2 27809.933} C_VEL
LIN {X 0,Y 37.533,Z 1276.599,A -85,B 0,C 180,E1 27863.451,E2 27863.451} C_VEL
LIN {X 0,Y 68.178,Z 1270.167,A -85,B 0,C 180,E1 27886.228,E2 27886.228} C_VEL
LIN {X 0,Y 102.228,Z 1258.376,A -85,B 0,C 180,E1 27894.956,E2 27894.956} C_VEL
LIN {X 0,Y 113.323,Z 1253.336,A -85,B 0,C 180,E1 27896.691,E2 27896.691} C_VEL
LIN {X 0,Y 79.305,Z 1267.92,A -85,B 0,C 180,E1 27903.003,E2 27903.003} C_VEL
LIN {X 0,Y 70.199,Z 1270.942,A -85,B 0,C 180,E1 27905.687,E2 27905.687} C_VEL
LIN {X 0,Y 53.469,Z 1275.207,A -85,B 0,C 180,E1 27908.522,E2 27908.522} C_VEL
LIN {X 0,Y 36.621,Z 1278.303,A -85,B 0,C 180,E1 27913.674,E2 27913.674} C_VEL
LIN {X 0,Y 16.042,Z 1281.185,A -85,B 0,C 180,E1 27970.185,E2 27970.185} C_VEL
LIN {X 0,Y 15.918,Z 1281.366,A -85,B 0,C 180,E1 27990.105,E2 27990.105} C_VEL
LIN {X 0,Y 31.876,Z 1279.106,A -85,B 0,C 180,E1 28061.394,E2 28061.394} C_VEL
LIN {X 0,Y 35.117,Z 1278.451,A -85,B 0,C 180,E1 28067.454,E2 28067.454} C_VEL
LIN {X 0,Y 37.674,Z 1276.743,A -85,B 0,C 180,E1 28099.165,E2 28099.165} C_VEL
LIN {X 0,Y 33.453,Z 1277.235,A -85,B 0,C 180,E1 28105.435,E2 28105.435} C_VEL
LIN {X 0,Y 16.857,Z 1278.865,A -85,B 0,C 180,E1 28169.901,E2 28169.901} C_VEL
LIN {X 0,Y 33.417,Z 1277.205,A -85,B 0,C 180,E1 28234.46,E2 28234.46} C_VEL
LIN {X 0,Y 67.885,Z 1270.492,A -85,B 0,C 180,E1 28253.207,E2 28253.207} C_VEL
LIN {X 0,Y 80.499,Z 1266.815,A -85,B 0,C 180,E1 28256.08,E2 28256.08} C_VEL
LIN {X 0,Y 60.354,Z 1273.016,A -85,B 0,C 180,E1 28261.502,E2 28261.502} C_VEL
LIN {X 0,Y 36.621,Z 1278.303,A -85,B 0,C 180,E1 28273.674,E2 28273.674} C_VEL
LIN {X 0,Y 24.358,Z 1279.848,A -85,B 0,C 180,E1 28282.233,E2 28282.233} C_VEL
LIN {X 0,Y 8.069,Z 1280.676,A -85,B 0,C 180,E1 28330.57,E2 28330.57} C_VEL
LIN {X 0,Y 7.905,Z 1280.736,A -85,B 0,C 180,E1 28346.431,E2 28346.431} C_VEL
LIN {X 0,Y 24.211,Z 1279.305,A -85,B 0,C 180,E1 28431.686,E2 28431.686} C_VEL
LIN {X 0,Y 26.856,Z 1278.85,A -85,B 0,C 180,E1 28436.26,E2 28436.26} C_VEL
LIN {X 0,Y 27.786,Z 1278.253,A -85,B 0,C 180,E1 28451.192,E2 28451.192} C_VEL
LIN {X 0,Y 24.886,Z 1278.504,A -85,B 0,C 180,E1 28456.797,E2 28456.797} C_VEL
LIN {X 0,Y 8.968,Z 1279.467,A -85,B 0,C 180,E1 28529.814,E2 28529.814} C_VEL
LIN {X 0,Y 36.725,Z 1277.106,A -85,B 0,C 180,E1 28611.359,E2 28611.359} C_VEL
LIN {X 0,Y 45.431,Z 1275.791,A -85,B 0,C 180,E1 28614.777,E2 28614.777} C_VEL
LIN {X 0,Y 45.297,Z 1275.937,A -85,B 0,C 180,E1 28617.196,E2 28617.196} C_VEL
LIN {X 0,Y 16.01,Z 1280.067,A -85,B 0,C 180,E1 28639.825,E2 28639.825} C_VEL
LIN {X 0,Y 7.905,Z 1280.736,A -85,B 0,C 180,E1 28706.431,E2 28706.431} C_VEL
LIN {X 0,Y 4.348,Z 1280.507,A -85,B 0,C 180,E1 28723.303,E2 28723.303} C_VEL
LIN {X 0,Y 1.079,Z 1280.069,A -85,B 0,C 180,E1 28888.454,E2 28888.454} C_VEL
LIN {X 0,Y 3.231,Z 1282.063,A -85,B 0,C 180,E1 28889.484,E2 28889.484} C_VEL
LIN {X 0,Y 3.231,Z 1319.5,A -85,B 0,C 180,E1 28889.484,E2 28889.484} C_VEL
LIN {X 0,Y 3.231,Z 1319.5,A -85,B 0,C 180,E1 28889.484,E2 28889.484}

